{attribute 'linkalways'} 
{attribute 'no_explicit_call' := 'This FB is a CLASS and must be accessed using methods or properties'}
{attribute 'enable_dynamic_creation'}
FUNCTION_BLOCK _LINT EXTENDS IntegerDatatypeBase
VAR
	localData : LINT;
	activeData : REFERENCE TO LINT REF= localData;
END_VAR

PROPERTY PUBLIC Address : PVOID
GET
Address := ADR(activeData);
END_GET
END_PROPERTY

METHOD PUBLIC ClearReference
VAR_INPUT
END_VAR
activeData REF= localData;
END_METHOD

METHOD PUBLIC Clone : I_Datatype
VAR
    pClone : POINTER TO _LINT;
END_VAR
pClone := __NEW(_LINT(InitialValue := Value));
Clone := pClone^;
END_METHOD

PROPERTY PUBLIC Datatype : T_MAXSTRING
GET
Datatype := 'LINT';
END_GET
END_PROPERTY

METHOD FB_init : BOOL
VAR_INPUT
	bInitRetains : BOOL; // if TRUE, the retain variables are initialized (warm start / cold start)
	bInCopyCode : BOOL;  // if TRUE, the instance afterwards gets moved into the copy code (online change)
	InitialValue : LINT;
END_VAR
localData := InitialValue;
END_METHOD

PROPERTY PUBLIC IsSigned : BOOL
GET
IsSigned := TRUE;
END_GET
END_PROPERTY

PROPERTY PUBLIC LowerBound : LINT
GET
LowerBound := DatatypeLimits.LINT_LOWER_LIMIT;
END_GET
END_PROPERTY

METHOD PUBLIC MakeReferenceTo
VAR_INPUT
	ReferenceTarget : REFERENCE TO LINT;
END_VAR
activeData REF= ReferenceTarget;
END_METHOD

METHOD PROTECTED SerializeLowerbound
VAR_INPUT
	Serializer : I_Serializer;
END_VAR
Serializer.AddLint(Lowerbound);
END_METHOD

METHOD PROTECTED SerializeUpperbound
VAR_INPUT
	Serializer : I_Serializer;
END_VAR
Serializer.AddLint(Upperbound);
END_METHOD

METHOD PUBLIC SerializeWith
VAR_INPUT
	Serializer : I_Serializer;
END_VAR
Serializer.AddLint(activeData);
END_METHOD

PROPERTY PUBLIC Size : UDINT
GET
Size := SIZEOF(activeData);
END_GET
END_PROPERTY

METHOD TryDeserializeFrom : BOOL
VAR_INPUT
	Deserializer : I_Deserializer;
	Feedback : I_DeserializerFeedback;
END_VAR
TryDeserializeFrom := Deserializer.TryGetLint(activeData, Feedback);
END_METHOD

METHOD TryMakeReferenceTo : BOOL
VAR_INPUT
	Target : I_Datatype;
END_VAR
VAR
	pTargetData : POINTER TO LINT;
END_VAR
IF NOT (Target.Datatype = Datatype) THEN
	RETURN;
END_IF

pTargetData := Target.Address;
activeData REF= pTargetData^;
TryMakeReferenceTo := TRUE;
END_METHOD

PROPERTY PUBLIC UpperBound : LINT
GET
UpperBound :=  DatatypeLimits.LINT_UPPER_LIMIT;
END_GET
END_PROPERTY

PROPERTY PUBLIC Value : LINT
GET
Value := activeData;
END_GET
SET
activeData := Value;
END_SET
END_PROPERTY

END_FUNCTION_BLOCK

(* stored: Version 1.1.0.1, ProductVersion 3.1.4024.12
   POU _LINT: Id {5bc7f1dd-5c23-04b5-2988-14762c8a8f8c}, SpecialFunc None
   Folder Constructor: Id {2e3dbac4-df59-0cfa-3714-defc8af50f7b}
   Folder Protected: Id {c3e95bf8-0859-043b-06b0-01464a9a08b6}
   Property Address: Id {0db9698f-71b2-0e3a-3f12-09e067e113ed}
   Get Get: Id {d8cd103f-bebd-04c0-1c90-c740ec1d1969}
   Method ClearReference: Id {d1aa4db9-004c-0671-37c1-fff8d7d96b41}
   Method Clone: Id {6741eddd-9143-0293-293d-2e3844335b8a}
   Property Datatype: Id {4f73e892-d305-03b1-3ff8-3c18c8f84cbd}
   Get Get: Id {f2d7ead6-7875-0053-38b9-740982899b2e}
   Method FB_init: Id {a4df2d97-2866-0f97-1768-ebcce6eac5de}
   Property IsSigned: Id {7eae4ba8-d49c-07bb-0355-55d0462e35fa}
   Get Get: Id {79b2931a-5bff-0a12-0cf2-6b9902ca1252}
   Property LowerBound: Id {ce54839e-2b96-0db3-0e8e-fc481b95b49b}
   Get Get: Id {c38796d3-283a-0711-0dcd-9af8c87f4905}
   Method MakeReferenceTo: Id {82af78ec-5741-0717-13be-6f12739589bb}
   Method SerializeLowerbound: Id {fd727f69-2ca1-0f1e-009c-3cf16d8643a9}
   Method SerializeUpperbound: Id {e3e7bc57-75e8-0519-38b4-a72f6e575901}
   Method SerializeWith: Id {1e289958-6813-057a-3a07-7d697036efce}
   Property Size: Id {9a1e20b5-4d86-0c7a-38e6-f8a10d38c5b3}
   Get Get: Id {6dc791f2-ee94-0866-1ff1-fe433a62a6eb}
   Method TryDeserializeFrom: Id {967ecf97-be61-0c36-1deb-a9d0dd8a2eff}
   Method TryMakeReferenceTo: Id {04756b22-6eae-0583-0e6d-4cdffd0edbdc}
   Property UpperBound: Id {4a66617a-b23b-0bf7-266e-1e05f6733294}
   Get Get: Id {76cd0108-4ea1-004e-32a2-4485c1dfafc9}
   Property Value: Id {fd15c92e-eab9-0007-0dfe-350b39f88ae7}
   Get Get: Id {21ef97a5-6387-0daf-19ae-c76b24796325}
   Set Set: Id {a0a5cb04-bc8e-0024-0792-f12f4ec25d04} *)
